// TIA Portal project "sps" (V16)

(* hardware
DEVICE "S7-1200-Station_1"  S7-1200 Station
   slot 0: "Baugruppenträger_0"  S7-1200 Rack  Rack  V1.0
   slot 1: "PLC_1"  CPU 1214C DC/DC/DC  6ES7 214-1AG40-0XB0  V4.4
*)

// ===== PLC "PLC_1"  CPU 1214C DC/DC/DC =====

VAR_GLOBAL   // PLC tag table "Standard-Variablentabelle"
   "OUT" AT %Q0.0 : Bool;
   "IN1" AT %I0.0 : Bool;
   "IN1.1" AT %I0.1 : Bool;
   "IN1.2" AT %I0.2 : Bool;
   "IN1.3" AT %I0.3 : Bool;
   "OUT1" AT %Q0.1 : Bool;
END_VAR

DATA_BLOCK "Datenbaustein_1"   // DB1
{ S7_Optimized_Access := 'FALSE' }
VERSION : 0.1
   VAR
      E00 : Bool;
      E01 : Bool;
      E02 : Bool;
      E03 : Bool;
      E04 : Bool;
      E05 : Bool;
      E06 : Bool;
      E07 : Bool;
      E10 : Bool;
      E11 : Bool;
      E12 : Bool;
      E13 : Bool;
      E14 : Bool;
      E15 : Bool;
      A00 : Bool;
      A01 : Bool;
      A02 : Bool;
      A03 : Bool;
      A04 : Bool;
      A05 : Bool;
      A06 : Bool;
      A07 : Bool;
      A10 : Bool;
      A11 : Bool;
   END_VAR
BEGIN
END_DATA_BLOCK

// folder: System blocks/Program resources

DATA_BLOCK "IEC_Timer_0_DB"   // DB2
{ S7_Optimized_Access := 'TRUE' }
AUTHOR : Simatic
FAMILY : IEC
NAME : IEC_TMR
VERSION : 1.0
// stored: InstanceOfName IEC_TIMER
"IEC_TIMER"
BEGIN
END_DATA_BLOCK

DATA_BLOCK "IEC_Timer_0_DB_1"   // DB3
{ S7_Optimized_Access := 'TRUE' }
AUTHOR : Simatic
FAMILY : IEC
NAME : IEC_TMR
VERSION : 1.0
// stored: InstanceOfName IEC_TIMER
"IEC_TIMER"
BEGIN
END_DATA_BLOCK

// folder: (top level)

ORGANIZATION_BLOCK "Main"   // OB1, FBD, ProgramCycle
TITLE = "Main Program Sweep (Cycle)"
{ S7_Optimized_Access := 'TRUE' }
VERSION : 0.1
   VAR_INPUT
      Initial_Call : Bool;   // Initial call of this OB
      Remanence : Bool;   // =True, if remanent data are available
   END_VAR
BEGIN

REGION Network 1
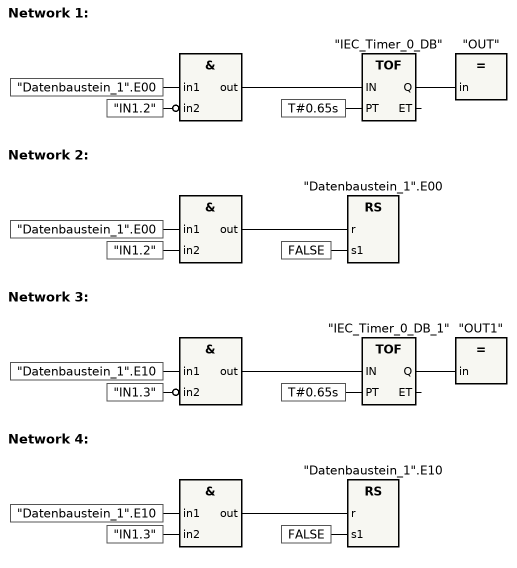
   "IEC_Timer_0_DB".TOF(IN := "Datenbaustein_1".E00 AND NOT "IN1.2", PT := T#0.65s);
   "OUT" := "IEC_Timer_0_DB".Q;
END_REGION

REGION Network 2
   IF "Datenbaustein_1".E00 AND "IN1.2" THEN
       "Datenbaustein_1".E00 := FALSE;   // RS flip-flop
   END_IF;
   IF FALSE THEN "Datenbaustein_1".E00 := TRUE; END_IF;
END_REGION

REGION Network 3
   "IEC_Timer_0_DB_1".TOF(IN := "Datenbaustein_1".E10 AND NOT "IN1.3", PT := T#0.65s);
   "OUT1" := "IEC_Timer_0_DB_1".Q;
END_REGION

REGION Network 4
   IF "Datenbaustein_1".E10 AND "IN1.3" THEN
       "Datenbaustein_1".E10 := FALSE;   // RS flip-flop
   END_IF;
   IF FALSE THEN "Datenbaustein_1".E10 := TRUE; END_IF;
END_REGION
END_ORGANIZATION_BLOCK